(* IEC 61131-3 sources: ICSQuartz/benchmarks/oscat_basic_fstring_to_byte/src, 1 file *)

(* ---- program.st ---- *)
PROGRAM PLC_PRG
VAR_INPUT
    in_in: STRING(12);
END_VAR

FSTRING_TO_BYTE(in_in);

END_PROGRAM
